// TIA Portal V17 export
// export: Created 2022-07-20T07:01:32.3263417Z, ExportSetting WithDefaults, DisplayName Totally Integrated Automation Portal, DisplayVersion V17, DisplayName TIA Portal Openness, DisplayVersion V17, DisplayName TIA Portal Version Control Interface, DisplayVersion V17, DisplayName SINAMICS Startdrive Advanced, DisplayVersion V17, DisplayName SINAMICS Startdrive G130, G150, S120, S150, SINAMICS MV, S210, DisplayVersion V17, DisplayName SINAMICS Startdrive G110M, G120, G120C, G120D, G120P, G115D, DisplayVersion V17, DisplayName STEP 7 Professional, DisplayVersion V17, DisplayName STEP 7 Safety, DisplayVersion V17, DisplayName WinCC Advanced, DisplayVersion V17
FUNCTION_BLOCK "FB10343_WinderFoil"   // FB10343, LAD
{ S7_Optimized_Access := 'TRUE' }
VERSION : 0.1
// stored: AutoNumber false, IsIECCheckEnabled false, IsRetainMemResEnabled false, MemoryReserve 100, SetENOAutomatically false, UDAEnableTagReadback false
   VAR_INPUT
      RequestAcknowledge : Bool;
      Ready : Bool;
   END_VAR
   VAR_OUTPUT
      ActiveWinder : Bool;
      WinderActivated : Bool;
      WinderInError : Bool;
      InverterStart : Bool;
   END_VAR
   VAR_IN_OUT
      RequestActiveWinder : Bool;
   END_VAR
   VAR
      R_TRIG_RequestActiveWinder : R_TRIG;
      F_TRIG_RequestActiveWinder { S7_SetPoint := 'True'} : F_TRIG;
      TON_WinderActivated { S7_SetPoint := 'True'} : TON_TIME;
      TON_WinderNotActivated { S7_SetPoint := 'True'} : TON_TIME;
      TON_WinderInError { S7_SetPoint := 'True'} : TON_TIME;
      TON_InverterStart { S7_SetPoint := 'True'} : TON_TIME;
   END_VAR
BEGIN

REGION Network 1 (SCL): First Scan
   IF "FirstScan" THEN
       #ActiveWinder := FALSE;
       #WinderActivated := FALSE;
       #InverterStart := FALSE;
   END_IF;
END_REGION

REGION Network 2 (SCL): Edge Signals & Timers
   REGION EDGE SIGNALS
       #R_TRIG_RequestActiveWinder(CLK := #RequestActiveWinder);

       #F_TRIG_RequestActiveWinder(CLK := #RequestActiveWinder);
   END_REGION ;

   REGION TIMERS
       #TON_WinderActivated(IN := #ActiveWinder,
                              PT := T#1s);
       #TON_WinderNotActivated(IN := NOT (#ActiveWinder),
                                 PT := T#1s);
       #TON_InverterStart(IN := #InverterStart,
                          PT := T#1s);
       #TON_WinderInError(IN := #RequestActiveWinder AND NOT (#ActiveWinder)
                            OR #RequestActiveWinder AND NOT (#WinderActivated)
                            OR NOT (#RequestActiveWinder) AND #ActiveWinder
                            OR NOT (#RequestActiveWinder) AND #WinderActivated,
                            PT := T#1s);
   END_REGION ;
END_REGION

REGION Network 3 (SCL): Unwinder Management
   IF #R_TRIG_RequestActiveWinder.Q THEN
       #ActiveWinder := TRUE;
   ELSIF #F_TRIG_RequestActiveWinder.Q THEN
       #ActiveWinder := FALSE;
   END_IF;
END_REGION

REGION Network 4 (SCL): States
   IF #TON_WinderActivated.Q THEN
       #WinderActivated := TRUE;
   ELSIF #TON_WinderNotActivated.Q THEN
       #WinderActivated := FALSE;
   END_IF;


   IF #TON_WinderInError.Q THEN
       #WinderInError := TRUE;
   ELSIF #RequestAcknowledge THEN
       #WinderInError := false;
   END_IF;

   IF #TON_InverterStart.Q THEN
       #InverterStart := TRUE;
   ELSIF #RequestAcknowledge THEN
       #InverterStart := FALSE;
   END_IF;
END_REGION
END_FUNCTION_BLOCK
